Staubli VAL3: message.pgx

public program message(string& message[], num index)
// Italian IF message
begin
  // lenght of message
  //
  switch index
    case 0
      message="Si vuole accedere all'interno del programma:"
    break
    case 1
      message="< Assistente IF >"
    break
    case 2
      message="Selezionare il tipo di condizione da verificare"
    break
    case 3
      message="Selezionare l'ingresso"
    break
    case 4
      message="Selezionare l'uscita"
    break
    case 5
      message="Selezionare l'ingresso EMAP"
    break
    case 6
      message="Selezionare come avviare l'istruzione"
    break
    case 7
      message="Selezionare l'istruzione da associare a: "
    break
    case 8
      message="Selezionare dalla lista "
    break
  endSwitch
end
